(********************************************************************************************)
(*							Beckhoff Automation Poland										*)
(*							F_Words_to_Real													*)
(*									12.05.2011												*)
(*			Funkcja składa dwie wartości typu WORD  i zamienia na watrosc typu REAL			*)
(*__________________________________________________________________________________________*)

FUNCTION F_Words_to_Real : REAL
VAR_INPUT
	wUpperWord : WORD;
	wLowerWord :WORD;
END_VAR
VAR
END_VAR

MEMCPY(ADR(F_Words_to_Real),ADR(wUpperWord),2);
MEMCPY(ADR(F_Words_to_Real)+2,ADR(wLowerWord),2);

END_FUNCTION

(* stored: Version 1.1.0.1, ProductVersion 3.1.4026.13, FileIdentifier 65b4532f73f3fdbc3aa24aaf3609ed685dbf527e, FileSignature 474d75ff287bf7817260ad56ad49a18eec21c45b4602cd7b74479e5f6c39d2dca8da7d0e045713940e12461cd03c46848cead2e6cf5aed6822b25110a885c3958cf2909c5db6d9f9bab4bed04ffd4c2152a02d6dd1aa94196bff39fb4831ab12eae7f2f98a111660f8f0182d2361b0a7a3e6f6fc221c7826e7f29ccb461925504ecc091e9312a1348093e20c2076c02ef987d8b478f3acc3cd26f2cc346b0be7863d3972084ebd00a4165c66b67d9ab7bc623634892f28fe126472fc209516cace6c6eb307e316d99109571e43055fcdc1ec1223694feba906c97489f8e46841d99cf7bf607cc5ea4a5ca036ef3d198287195e69da2cfaa16b9bbbe0758ef9a3
   POU F_Words_to_Real: Id {4b7d83e9-860f-4642-8220-e277b0168541}, SpecialFunc None *)
